FUNCTION F_vltMod : LREAL
VAR_INPUT
	number:		LREAL;
	divisor:	LREAL;
END_VAR
VAR
END_VAR

(*
static double vltMod(double number, double divisor)
{
    if (divisor == 0.0)
	return 0.0;
    return number - divisor * (int) (number / divisor);
}


*)

IF divisor = 0.0 THEN
	F_vltMod	:= 0.0;
ELSE
	F_vltMod	:= number - divisor * TRUNC_INT(number / divisor);
END_IF

END_FUNCTION

(* stored: Version 1.1.0.1, ProductVersion 3.1.4022.9
   POU F_vltMod: Id {fde37526-7a6e-4770-9cc9-4baa0770a045}, SpecialFunc None *)
